Yaskawa INFORM job: X4-SCHODKI_ZEW.JBI

/JOB
//NAME X4-SCHODKI_ZEW
//POS
///NPOS 247,247,247,10,0,0
///TOOL 0
///POSTYPE PULSE
///PULSE
C00000=-21160,-126487,-99095,-6220,53097,-19917
C00001=-122314,-84956,-84267,-5758,65294,-20346
C00002=-113867,-2788,-32259,-11364,77586,20622
C00003=-111699,9606,-11794,-12514,71800,21939
C00004=-110873,16102,-4909,-12893,71047,22311
C00005=-111426,18220,-2948,-12689,70847,22135
C00006=-111334,17863,-3281,-12723,70881,22164
C00007=-111334,17842,-1921,-12786,70054,22254
C00008=-111688,13758,-7042,-12574,71029,22022
C00009=-137921,23655,2193,26065,80546,-13065
C00010=-138187,30095,8478,26164,80127,-13260
C00011=-137141,31636,10013,25924,79665,-12972
C00012=-137283,31426,9804,25956,79727,-13011
C00013=-137283,31447,11085,26011,79025,-13166
C00014=-137811,24810,3269,26040,80453,-13045
C00015=-130093,15204,-5597,17076,73087,-3422
C00016=-130254,16762,-4164,17139,73044,-3486
C00017=-130499,11823,-8660,17205,73314,-3535
C00018=-136657,16032,-4835,19303,74485,-5576
C00019=-136779,34044,12201,19450,73350,-5806
C00020=-136367,37287,16065,19383,72578,-5782
C00021=-135529,38270,17077,19116,72272,-5524
C00022=-135735,38345,17156,19186,72312,-5593
C00023=-135735,38391,18179,19247,71738,-5687
C00024=-136093,38073,17157,19317,72259,-5733
C00025=-136821,38987,18103,19565,72324,-5991
C00026=-137234,41236,20445,19732,72152,-6174
C00027=-137468,37941,16529,19737,72884,-6137
C00028=-139273,33119,8814,10616,74138,-14432
C00029=-138400,39162,15428,10360,73077,-14220
C00030=-137624,40756,17090,10099,72782,-13973
C00031=-137810,40443,16764,10163,72844,-14033
C00032=-137810,40460,18419,10216,71849,-14119
C00033=-138377,33107,10032,10341,73283,-14197
C00034=-129933,32626,9546,-1459,71562,-3103
C00035=-130107,34413,11352,-1398,71367,-3162
C00036=-130344,28976,5916,-1305,71915,-3250
C00037=-134876,30968,7890,396,71698,-4822
C00038=-142592,70732,50995,12851,68399,-16892
C00039=-141830,71409,51797,12602,68137,-16639
C00040=-142006,70894,51186,12652,68274,-16689
C00041=-142006,71149,52557,12712,67578,-16765
C00042=-142006,71007,51815,12679,67954,-16725
C00043=-142747,76515,58410,13043,66871,-17119
C00044=-142702,66110,44987,12780,69711,-16790
C00045=-130401,22900,-3912,-9781,74013,-14096
C00046=-130750,-77898,-76934,-10038,67211,-13654
C00047=-128341,-94500,-64478,-15665,37561,-8814
C00048=-125354,-34494,-33676,-16070,41961,-8103
C00049=-123908,-22688,-35224,7311,60763,-8117
C00050=-115329,1774,-22996,8583,68206,-33205
C00051=-113811,6923,-16554,7934,66753,-32769
C00052=-112938,8598,-15088,7517,66630,-32466
C00053=-113357,7607,-15958,7718,66694,-32611
C00054=-113357,7474,-14642,7767,65823,-32669
C00055=-113357,7562,-15559,7732,66427,-32629
C00056=-114674,8046,-17033,9196,71995,-10105
C00057=-114277,9137,-16073,9034,71921,-9973
C00058=-114994,10710,-14679,9331,71949,-10219
C00059=-115929,5782,-19714,10610,72890,-11247
C00060=-114914,9168,-18033,20160,83408,-25507
C00061=-114509,10465,-16323,20060,82947,-25443
C00062=-114509,10278,-15209,20089,82211,-25564
C00063=-114509,10430,-16126,20066,82816,-25464
C00064=-113574,12027,-14696,19812,82540,-25184
C00065=-113966,9476,-16971,19916,82715,-25292
C00066=-109195,41890,2270,19889,88323,-22522
C00067=-109420,41611,2136,14547,83651,-24420
C00068=-109633,43097,3705,14621,83493,-24508
C00069=-110073,47498,8361,9922,80898,-20177
C00070=-110340,48514,8983,10012,81065,-20250
C00071=-109875,50139,10594,6927,80049,-17487
C00072=-111642,41129,-2073,7513,83338,-17864
C00073=-120740,-4591,-30289,15267,55452,-23675
C00074=-120758,-111403,-89341,20679,37744,-27189
C00075=-120758,-111403,-89341,20679,37744,-27189
C00076=-97140,-41370,-74515,-11864,90116,15742
C00077=-93918,-16818,-51601,-15265,90472,19448
C00078=-96838,-21310,-54909,-14446,89719,18600
C00079=-97144,-22320,-55662,-14359,89616,18514
C00080=-98771,-24881,-57497,-13895,89173,18041
C00081=-115828,-29996,-61044,7286,86100,-2495
C00082=-121364,-24267,-57094,13933,89260,-9154
C00083=-125064,-13370,-49143,14990,90552,-10191
C00084=-125209,-12228,-48362,15033,90681,-10222
C00085=-127775,-3453,-41245,15747,91251,-10973
C00086=-117906,-11103,-47413,1372,86513,3179
C00087=-107817,-4833,-42392,-13913,90158,17947
C00088=-111065,-8601,-45456,-12965,89620,16971
C00089=-111228,-9142,-45834,-12917,89553,16926
C00090=-113235,-11504,-47787,-12324,89257,16321
C00091=-116129,-16038,-53218,-11461,89860,15351
C00092=-132129,3503,-37461,-731,88042,5165
C00093=-134330,9298,-30541,1308,86617,3236
C00094=-133591,9704,-30242,1064,86631,3463
C00095=-133365,10194,-29830,989,86627,3533
C00096=-132997,13157,-27039,5636,86965,-851
C00097=-131112,-12606,-50888,7793,88905,-29033
C00098=-129834,-10886,-48018,7386,87922,-28697
C00099=-133242,1411,-38107,8469,88444,-29724
C00100=-133268,2556,-37251,8479,88508,-29727
C00101=-132895,14601,-26523,2898,86979,-24450
C00102=-133144,15447,-25750,2979,86944,-24527
C00103=-133588,9909,-35564,3125,90148,-24585
C00104=-114600,-38617,-66572,-24501,76796,-21744
C00105=-88804,-102668,-113384,-34072,81784,-13502
C00106=3643,-76224,-106676,19950,71810,76872
C00107=6047,-95755,-92046,-14751,98253,9605
C00108=8024,-164446,-133802,-16041,6272,12396
C00109=8024,-164446,-133802,-16041,6272,12396
C00110=80911,-131071,-112390,-19160,57527,-4768
C00111=107387,-112645,-89313,-18613,48039,-3448
C00112=120529,-94925,-67119,-18087,38914,-2179
C00113=119158,-22093,-21003,-8683,62714,-5793
C00114=120616,-13235,-11129,-9376,61371,-5124
C00115=120244,-10241,-8815,-9223,61441,-5272
C00116=120242,-11093,-9478,-9225,61411,-5270
C00117=120242,-10458,-7028,-9331,60244,-5174
C00118=120224,-17007,-14555,-9215,61493,-5286
C00119=122889,-18524,910,-53470,54044,-6110
C00120=122847,-15690,3005,-53366,54123,-6195
C00121=122811,-12986,5045,-53281,54183,-6262
C00122=122821,-13724,4484,-53302,54168,-6245
C00123=122821,-12957,6355,-53740,53705,-5906
C00124=125895,-21581,-2992,-53539,56263,-5738
C00125=123923,-36868,-26996,-37261,61302,-5894
C00126=108816,-52753,-53811,-10212,62008,-9374
C00127=96034,-45136,-47055,9675,61622,-25160
C00128=97205,-43220,-45890,9111,61748,-24699
C00129=96974,-43470,-46044,9221,61740,-24787
C00130=96974,-43222,-44278,9303,60791,-24865
C00131=96448,-45521,-47615,9470,61714,-24990
C00132=118629,-40101,-48504,-12157,74776,12413
C00133=119364,-34097,-44083,-12359,75244,12623
C00134=118100,-32224,-42841,-11965,75251,12181
C00135=118253,-32582,-43080,-12015,75236,12237
C00136=118253,-32540,-41664,-12057,74406,12319
C00137=118721,-32602,-42752,-12165,75101,12411
C00138=116137,-37716,-46090,-11401,74165,11593
C00139=108993,-39238,-47060,-3979,71836,3847
C00140=109761,-37600,-46019,-4238,72074,4108
C00141=108993,-39238,-47060,-3979,71836,3847
C00142=117414,-43467,-49690,-6866,71847,6805
C00143=120406,-23125,-36428,-7781,74390,7697
C00144=120412,-21128,-34805,-7781,74419,7698
C00145=119620,-19753,-33804,-7516,74437,7425
C00146=119849,-20298,-34202,-7592,74423,7506
C00147=119849,-20300,-33096,-7616,73750,7551
C00148=119849,-20302,-33703,-7602,74119,7528
C00149=120845,-19874,-33391,-7929,74241,7866
C00150=121446,-18122,-32105,-8123,74405,8066
C00151=121464,-22241,-35587,-8130,74432,8070
C00152=122270,-32243,-42159,4732,69932,24573
C00153=121378,-24903,-37120,5049,70656,24286
C00154=120376,-23507,-36128,5424,70830,23939
C00155=120533,-24190,-36613,5366,70768,23993
C00156=120533,-24175,-35602,5386,70155,23966
C00157=120148,-30314,-42064,5504,71001,23867
C00158=110805,-25383,-38662,15109,74916,14576
C00159=111818,-22665,-36734,14771,74934,14940
C00160=111748,-27369,-40047,14817,74581,14871
C00161=119775,-28434,-40781,12151,73173,17551
C00162=124224,-1084,-19915,10540,73751,19166
C00163=130157,198,-18683,-209,73628,24476
C00164=130157,158,-17341,-210,72780,24477
C00165=130157,185,-18394,-210,73442,24477
C00166=129196,1421,-17357,132,73439,24146
C00167=130157,185,-18394,-210,73442,24477
C00168=122787,3680,-15441,12656,76349,11624
C00169=123743,5439,-13926,12357,76179,11938
C00170=123109,1410,-18093,12531,76759,11776
C00171=126751,-18741,-32489,13679,66636,29547
C00172=131594,-6512,-22252,11541,65879,31250
C00173=135627,-1986,-17513,3780,65616,32121
C00174=135627,-1956,-16347,3801,64914,32097
C00175=135627,-1986,-17486,3780,65599,32120
C00176=134800,-891,-16582,4152,65645,31822
C00177=135627,-1986,-17486,3780,65599,32120
C00178=122949,-12611,-24589,22132,67603,15841
C00179=121506,-8744,-21577,22663,68115,15387
C00180=122081,-6475,-19773,22437,68011,15585
C00181=121506,-8744,-21577,22663,68115,15387
C00182=127706,-12999,-26066,20142,67056,17565
C00183=136075,11793,-4386,8081,62286,35157
C00184=136075,11856,-3257,8130,61628,35109
C00185=136075,11798,-4304,8086,62236,35152
C00186=136366,13707,-2741,6760,62424,35173
C00187=136075,11798,-4304,8086,62236,35152
C00188=131305,-10305,-23416,10361,63176,33430
C00189=168291,-111367,-82610,-9688,47305,48503
C00190=206286,-74639,-65979,-25452,64014,61826
C00191=159660,-110455,-93035,-14572,38895,45711
C00192=139772,-9678,-45421,-20416,66544,-77404
C00193=128522,-26109,-48700,-36268,57340,-84657
C00194=119767,-9340,-33749,-20588,54929,-87055
C00195=118381,-12869,-36453,-19680,54464,-87541
C00196=118069,-13852,-36761,-19540,54093,-87599
C00197=119978,-17814,-39706,-30625,59015,-81414
C00198=119898,-18805,-40392,-30604,58911,-81418
C00199=117451,-25837,-45359,-31771,59062,-80695
C00200=122977,-25509,-47564,-34287,62428,-79397
C00201=137466,-21144,-46854,-40649,69913,-75869
C00202=196853,-39310,-56838,-56279,98183,-62272
C00203=239125,-37728,-55833,-56309,98295,-62347
C00204=198880,-64017,-70083,-47949,71692,22240
C00205=95782,-63494,-66422,9583,64100,-25040
C00206=96608,-32442,-40990,7123,69750,-24476
C00207=99153,-41436,-44893,7278,64322,-23821
C00208=98934,-42045,-45261,7777,64334,-23890
C00209=100370,-44106,-46526,7182,63922,-23380
C00210=119741,-40174,-44096,-19149,69535,-259
C00211=121592,-27553,-38534,-18093,79240,10876
C00212=125227,-17250,-31142,-18927,80757,11935
C00213=125393,-15914,-30142,-18963,80861,11977
C00214=127846,-8061,-24015,-19516,81680,12716
C00215=119795,-17677,-31449,-8017,74335,-710
C00216=108325,-15786,-29976,9492,74890,-18554
C00217=111630,-19800,-33189,8434,74445,-17438
C00218=111755,-20573,-33754,8397,74383,-17399
C00219=113687,-22438,-34957,7772,73974,-16756
C00220=117056,-24250,-37509,6639,74313,-15568
C00221=128480,-979,-19969,3779,76440,-7427
C00222=129844,2675,-15882,3356,75744,-6982
C00223=129268,3108,-15627,2949,75760,-6545
C00224=129028,3528,-15269,3025,75765,-6627
C00225=129576,5579,-13546,-2876,75741,-370
C00226=130057,-3886,-22978,-3018,76699,-230
C00227=122913,-28792,-41505,-1480,73376,7564
C00228=125274,-18849,-33719,-4896,77191,17730
C00229=131975,-10313,-25549,-10610,74903,19808
C00230=132069,-9167,-24748,-10635,75011,19832
C00231=135966,6668,-11544,-11862,75556,21141
C00232=130236,2592,-15119,-2350,73160,11427
C00233=128403,-11609,-30449,-1692,75251,10764
C00234=112588,-48510,-57222,11111,73491,6010
C00235=118900,-27089,-23855,-4947,60648,-6067
C00236=130292,-938,239,-22775,68727,4409
C00237=117379,-19874,-3208,-40401,48526,-8648
C00238=111452,-18537,-670,-42583,47269,-4687
C00239=115600,-23691,-9256,-36668,53200,-7502
C00240=123114,-34014,-31898,-14023,63529,-7414
C00241=103776,-61917,-65189,16989,73535,3120
C00242=77625,-115928,-93453,24842,70557,-7280
C00243=80911,-131071,-112390,-19160,57527,-4768
C00244=8024,-164446,-133802,-16041,6272,12396
C00245=8024,-164446,-133802,-16041,6272,12396
C00246=3643,-76224,-106676,19950,71810,76872
BC00000=277659,673923,172124
BC00001=328197,693320,172124
BC00002=328196,693321,172121
BC00003=328196,693321,172121
BC00004=328196,693321,172121
BC00005=328196,693321,172121
BC00006=328196,693321,172121
BC00007=328196,693321,172121
BC00008=328196,693321,172121
BC00009=328196,693321,172121
BC00010=328196,693321,172121
BC00011=328196,693321,172121
BC00012=328196,693321,172121
BC00013=328196,693321,172121
BC00014=328196,693321,172121
BC00015=328196,693321,172121
BC00016=328196,693321,172121
BC00017=328196,693321,172121
BC00018=328196,693321,172121
BC00019=328196,693321,172121
BC00020=328196,693321,172121
BC00021=328196,693321,172121
BC00022=328196,693321,172121
BC00023=328196,693321,172121
BC00024=328196,693321,172121
BC00025=328196,693321,172121
BC00026=328196,693321,172121
BC00027=328196,693321,172121
BC00028=328196,693321,172121
BC00029=328196,693321,172121
BC00030=328196,693321,172121
BC00031=328196,693321,172121
BC00032=328196,693321,172121
BC00033=328196,693321,172121
BC00034=328196,693321,172121
BC00035=328196,693321,172121
BC00036=328196,693321,172121
BC00037=328196,693321,172121
BC00038=328196,693321,172121
BC00039=328196,693321,172121
BC00040=328196,693321,172121
BC00041=328196,693321,172121
BC00042=328196,693321,172121
BC00043=328196,693321,172121
BC00044=328196,693321,172121
BC00045=328196,693321,172121
BC00046=328196,693321,172121
BC00047=194432,688081,172121
BC00048=194432,688081,172121
BC00049=173327,765103,172121
BC00050=173327,765103,140855
BC00051=173327,765103,140855
BC00052=173327,765103,140855
BC00053=173327,765103,140855
BC00054=173327,765103,140855
BC00055=173327,765103,140855
BC00056=173327,765103,140855
BC00057=173327,765103,140855
BC00058=173327,765103,140855
BC00059=173327,765103,140855
BC00060=173327,765103,140855
BC00061=173327,765103,140855
BC00062=173327,765103,140855
BC00063=173327,765103,140855
BC00064=173327,765103,140855
BC00065=173327,765103,140855
BC00066=158508,737843,59363
BC00067=158508,737843,59363
BC00068=158508,737843,59363
BC00069=158508,737843,59363
BC00070=158508,737843,59363
BC00071=158508,737843,59363
BC00072=158508,737843,59363
BC00073=158508,737843,59363
BC00074=158508,682152,59363
BC00075=293322,682152,59363
BC00076=293321,752433,59360
BC00077=293321,752433,59360
BC00078=293321,752433,59360
BC00079=293321,752433,59360
BC00080=293321,752433,59360
BC00081=293321,752433,59360
BC00082=293321,752433,59360
BC00083=293321,752433,59360
BC00084=293321,752433,59360
BC00085=293321,752433,59360
BC00086=293321,752433,59360
BC00087=293321,752433,59360
BC00088=293321,752433,59360
BC00089=293321,752433,59360
BC00090=293321,752433,59360
BC00091=293321,752433,59360
BC00092=293321,752433,59360
BC00093=293321,752433,59360
BC00094=293321,752433,59360
BC00095=293321,752433,59360
BC00096=293321,752433,59360
BC00097=293321,752433,59360
BC00098=293321,752433,59360
BC00099=293321,752433,59360
BC00100=293321,752433,59360
BC00101=293321,752433,59360
BC00102=293321,752433,59360
BC00103=293321,752433,59360
BC00104=293321,752433,59360
BC00105=293321,698561,59360
BC00106=199464,674570,1075173
BC00107=95044,675039,919146
BC00108=95044,675039,1075229
BC00109=235813,1345575,1075229
BC00110=291733,1363613,501241
BC00111=295042,1365829,344881
BC00112=288108,1367960,194507
BC00113=288108,1367960,194507
BC00114=288108,1367960,194507
BC00115=288108,1367960,194507
BC00116=288108,1367960,194507
BC00117=288108,1367960,194507
BC00118=288108,1367960,194507
BC00119=288108,1367960,194507
BC00120=288108,1367960,194507
BC00121=288108,1367960,194507
BC00122=288108,1367960,194507
BC00123=288108,1367960,194507
BC00124=288108,1367960,194507
BC00125=288108,1367445,194507
BC00126=288108,1366688,194507
BC00127=288109,1366690,194504
BC00128=288109,1366690,194504
BC00129=288109,1366690,194504
BC00130=288109,1366690,194504
BC00131=288109,1366690,194504
BC00132=288109,1366690,194504
BC00133=288109,1366690,194504
BC00134=288109,1366690,194504
BC00135=288109,1366690,194504
BC00136=288109,1366690,194504
BC00137=288109,1366690,194504
BC00138=288109,1366690,194504
BC00139=288109,1366690,194504
BC00140=288109,1366690,194504
BC00141=288109,1366690,194504
BC00142=288109,1366690,194504
BC00143=288109,1366690,194504
BC00144=288109,1366690,194504
BC00145=288109,1366690,194504
BC00146=288109,1366690,194504
BC00147=288109,1366690,194504
BC00148=288109,1366690,194504
BC00149=288109,1366690,194504
BC00150=288109,1366690,194504
BC00151=288109,1366690,194504
BC00152=288109,1366690,194504
BC00153=288109,1366690,194504
BC00154=288109,1366690,194504
BC00155=288109,1366690,194504
BC00156=288109,1366690,194504
BC00157=288109,1366690,194504
BC00158=288109,1366690,194504
BC00159=288109,1366690,194504
BC00160=288109,1366690,194504
BC00161=288109,1366690,194504
BC00162=288109,1366690,194504
BC00163=288109,1366690,194504
BC00164=288109,1366690,194504
BC00165=288109,1366690,194504
BC00166=288109,1366690,194504
BC00167=288109,1366690,194504
BC00168=288109,1366690,194504
BC00169=288109,1366690,194504
BC00170=288109,1366690,194504
BC00171=288109,1366690,194504
BC00172=288109,1366690,194504
BC00173=288109,1366690,194504
BC00174=288109,1366690,194504
BC00175=288109,1366690,194504
BC00176=288109,1366690,194504
BC00177=288109,1366690,194504
BC00178=288109,1366690,194504
BC00179=288109,1366690,194504
BC00180=288109,1366690,194504
BC00181=288109,1366690,194504
BC00182=288109,1366690,194504
BC00183=288109,1366690,194504
BC00184=288109,1366690,194504
BC00185=288109,1366690,194504
BC00186=288109,1366690,194504
BC00187=288109,1366690,194504
BC00188=288109,1366690,194504
BC00189=362373,1366690,194504
BC00190=212912,1366690,52238
BC00191=212912,1366690,52238
BC00192=212912,1366690,52238
BC00193=181372,1351458,52238
BC00194=181372,1351458,52238
BC00195=181372,1351458,52238
BC00196=181372,1351458,52238
BC00197=181372,1351458,52238
BC00198=181372,1351458,52238
BC00199=181372,1351458,52238
BC00200=181372,1351458,52238
BC00201=181372,1351458,52238
BC00202=258948,1351458,52238
BC00203=397724,1351458,84656
BC00204=397724,1351458,84656
BC00205=288109,1366690,194504
BC00206=288109,1366690,194504
BC00207=288109,1366690,194504
BC00208=288109,1366690,194504
BC00209=288109,1366690,194504
BC00210=288109,1366690,194504
BC00211=288109,1366690,194504
BC00212=288109,1366690,194504
BC00213=288109,1366690,194504
BC00214=288109,1366690,194504
BC00215=288109,1366690,194504
BC00216=288109,1366690,194504
BC00217=288109,1366690,194504
BC00218=288109,1366690,194504
BC00219=288109,1366690,194504
BC00220=288109,1366690,194504
BC00221=288109,1366690,194504
BC00222=288109,1366690,194504
BC00223=288109,1366690,194504
BC00224=288109,1366690,194504
BC00225=288109,1366690,194504
BC00226=288109,1366690,194504
BC00227=288109,1366690,194504
BC00228=288109,1366690,194504
BC00229=288109,1366690,194504
BC00230=288109,1366690,194504
BC00231=288109,1366690,194504
BC00232=288109,1366690,194504
BC00233=288109,1366690,194504
BC00234=288109,1366690,194504
BC00235=288109,1366690,194504
BC00236=288109,1366690,194504
BC00237=288109,1366690,194504
BC00238=288109,1366690,194504
BC00239=288109,1366690,194504
BC00240=288109,1366690,194504
BC00241=288109,1366690,194504
BC00242=288109,1366690,194504
BC00243=269895,1363613,501241
BC00244=235813,1345575,1075229
BC00245=95044,675039,1075229
BC00246=199464,674570,1075173
EC00000=-798156,0
EC00001=-798156,0
EC00002=-798153,-1
EC00003=-798153,-1
EC00004=-798153,-1
EC00005=-798153,-1
EC00006=-798153,-1
EC00007=-798153,-1
EC00008=-798153,-1
EC00009=-798153,-1
EC00010=-798153,-1
EC00011=-798153,-1
EC00012=-798153,-1
EC00013=-798153,-1
EC00014=-798153,-1
EC00015=-798153,-1
EC00016=-798153,-1
EC00017=-798153,-1
EC00018=-798153,-1
EC00019=-798153,-1
EC00020=-798153,-1
EC00021=-798153,-1
EC00022=-798153,-1
EC00023=-798153,-1
EC00024=-798153,-1
EC00025=-798153,-1
EC00026=-798153,-1
EC00027=-798153,-1
EC00028=-798153,-1
EC00029=-798153,-1
EC00030=-798153,-1
EC00031=-798153,-1
EC00032=-798153,-1
EC00033=-798153,-1
EC00034=-798153,-1
EC00035=-798153,-1
EC00036=-798153,-1
EC00037=-798153,-1
EC00038=-798153,-1
EC00039=-798153,-1
EC00040=-798153,-1
EC00041=-798153,-1
EC00042=-798153,-1
EC00043=-798153,-1
EC00044=-798153,-1
EC00045=-798153,-1
EC00046=-798153,-1
EC00047=-798153,-1
EC00048=-798153,-1
EC00049=-798153,-1
EC00050=-798153,-1
EC00051=-798153,-1
EC00052=-798153,-1
EC00053=-798153,-1
EC00054=-798153,-1
EC00055=-798153,-1
EC00056=-798153,-1
EC00057=-798153,-1
EC00058=-798153,-1
EC00059=-798153,-1
EC00060=-798153,-1
EC00061=-798153,-1
EC00062=-798153,-1
EC00063=-798153,-1
EC00064=-798153,-1
EC00065=-798153,-1
EC00066=-798153,-1
EC00067=-798153,-1
EC00068=-798153,-1
EC00069=-798153,-1
EC00070=-798153,-1
EC00071=-798153,-1
EC00072=-798153,-1
EC00073=-798153,-1
EC00074=-798153,-1
EC00075=-798153,-1
EC00076=-798151,-2
EC00077=-798151,-2
EC00078=-798151,-2
EC00079=-798151,-2
EC00080=-798151,-2
EC00081=-798151,-2
EC00082=-798151,-2
EC00083=-798151,-2
EC00084=-798151,-2
EC00085=-798151,-2
EC00086=-798151,-2
EC00087=-798151,-2
EC00088=-798151,-2
EC00089=-798151,-2
EC00090=-798151,-2
EC00091=-798151,-2
EC00092=-798151,-2
EC00093=-798151,-2
EC00094=-798151,-2
EC00095=-798151,-2
EC00096=-798151,-2
EC00097=-798151,-2
EC00098=-798151,-2
EC00099=-798151,-2
EC00100=-798151,-2
EC00101=-798151,-2
EC00102=-798151,-2
EC00103=-798151,-2
EC00104=-798151,-2
EC00105=-798151,-2
EC00106=-798151,-2
EC00107=-798156,0
EC00108=798156,0
EC00109=798156,0
EC00110=798156,0
EC00111=798156,0
EC00112=798156,0
EC00113=798156,0
EC00114=798156,0
EC00115=798156,0
EC00116=798156,0
EC00117=798156,0
EC00118=798156,0
EC00119=798156,0
EC00120=798156,0
EC00121=798156,0
EC00122=798156,0
EC00123=798156,0
EC00124=798156,0
EC00125=798156,0
EC00126=798156,0
EC00127=798155,0
EC00128=798155,0
EC00129=798155,0
EC00130=798155,0
EC00131=798155,0
EC00132=798155,0
EC00133=798155,0
EC00134=798155,0
EC00135=798155,0
EC00136=798155,0
EC00137=798155,0
EC00138=798155,0
EC00139=798155,0
EC00140=798155,0
EC00141=798155,0
EC00142=798155,0
EC00143=798155,0
EC00144=798155,0
EC00145=798155,0
EC00146=798155,0
EC00147=798155,0
EC00148=798155,0
EC00149=798155,0
EC00150=798155,0
EC00151=798155,0
EC00152=798155,0
EC00153=798155,0
EC00154=798155,0
EC00155=798155,0
EC00156=798155,0
EC00157=798155,0
EC00158=798155,0
EC00159=798155,0
EC00160=798155,0
EC00161=798155,0
EC00162=798155,0
EC00163=798155,0
EC00164=798155,0
EC00165=798155,0
EC00166=798155,0
EC00167=798155,0
EC00168=798155,0
EC00169=798155,0
EC00170=798155,0
EC00171=798155,0
EC00172=798155,0
EC00173=798155,0
EC00174=798155,0
EC00175=798155,0
EC00176=798155,0
EC00177=798155,0
EC00178=798155,0
EC00179=798155,0
EC00180=798155,0
EC00181=798155,0
EC00182=798155,0
EC00183=798155,0
EC00184=798155,0
EC00185=798155,0
EC00186=798155,0
EC00187=798155,0
EC00188=798155,0
EC00189=798155,0
EC00190=798155,0
EC00191=798155,0
EC00192=798155,0
EC00193=798155,0
EC00194=798155,0
EC00195=798155,0
EC00196=798155,0
EC00197=798155,0
EC00198=798155,0
EC00199=798155,0
EC00200=798155,0
EC00201=798155,0
EC00202=798155,0
EC00203=798155,0
EC00204=798155,0
EC00205=798155,0
EC00206=798155,0
EC00207=798155,0
EC00208=798155,0
EC00209=798155,0
EC00210=798155,0
EC00211=798155,0
EC00212=798155,0
EC00213=798155,0
EC00214=798155,0
EC00215=798155,0
EC00216=798155,0
EC00217=798155,0
EC00218=798155,0
EC00219=798155,0
EC00220=798155,0
EC00221=798155,0
EC00222=798155,0
EC00223=798155,0
EC00224=798155,0
EC00225=798155,0
EC00226=798155,0
EC00227=798155,0
EC00228=798155,0
EC00229=798155,0
EC00230=798155,0
EC00231=798155,0
EC00232=798155,0
EC00233=798155,0
EC00234=798155,0
EC00235=798155,0
EC00236=798155,0
EC00237=798155,0
EC00238=798155,0
EC00239=798155,0
EC00240=798155,0
EC00241=798155,0
EC00242=798155,0
EC00243=798156,0
EC00244=798156,0
EC00245=798156,0
EC00246=798156,0
///POSTYPE BASE
///RECTAN
///RCONF 0,0,0,0,0,0,0,0,0,0,0,0,0,0,0,0,0,0,0,0,0,0,0,0
P00006=0.000,0.000,0.000,0.0000,0.0000,0.0000
P00021=1.195,-1.322,-3.236,0.0000,0.0000,0.0000
P00022=0.222,-3.123,-1.508,0.0000,0.0000,0.0000
P00023=0.143,-0.036,0.682,0.0000,0.0000,0.0000
P00024=0.145,-0.552,1.326,0.0000,0.0000,0.0000
P00025=-2.003,0.006,0.728,0.0000,0.0000,0.0000
P00026=0.562,-0.002,-0.337,0.0000,0.0000,0.0000
P00027=-0.746,0.015,-9.096,0.0000,0.0000,0.0000
P00030=5.926,-4.294,-1.390,0.0000,0.0000,0.0000
P00031=1.853,-0.001,-1.549,0.0000,0.0000,0.0000
//INST
///DATE 2024/04/14 21:21
///ATTR SC,RW
///GROUP1 RB1,BS1
///GROUP2 ST1
NOP
MOVJ C00000 BC00000 VJ=100.00  +MOVJ EC00000 VJ=100.00
MOVJ C00001 BC00001 VJ=100.00  +MOVJ EC00001 VJ=100.00
MOVJ C00002 BC00002 VJ=100.00  +MOVJ EC00002 VJ=100.00
SMOVL C00003 BC00003 V=833.3  +MOVJ EC00003
SMOVL C00004 BC00004 V=166.7  +MOVJ EC00004
SREFP 3 C00005 BC00005  +REFP EC00005
CALL JOB:SEARCH-R1-S13D
SET P021 P006
SFTON3D P021
SMOVL C00006 BC00006 V=166.7  +MOVJ EC00006
SREFP 3 C00007 BC00007  +REFP EC00007
CALL JOB:SEARCH-R1-S13D
SET P021 P006
SFTON3D P021
SMOVL C00008 BC00008 V=166.7  +MOVJ EC00008
SFTOF3D
SMOVL C00009 BC00009 V=833.3  +MOVJ EC00009
SMOVL C00010 BC00010 V=166.7  +MOVJ EC00010
SREFP 3 C00011 BC00011  +REFP EC00011
CALL JOB:SEARCH-R1-S13D
SET P022 P006
SFTON3D P022
SMOVL C00012 BC00012 V=166.7  +MOVJ EC00012
SREFP 3 C00013 BC00013  +REFP EC00013
CALL JOB:SEARCH-R1-S13D
SET P022 P006
SFTON3D P022
SMOVL C00014 BC00014 V=166.7  +MOVJ EC00014
SMOVL C00015 BC00015 V=166.7  +MOVJ EC00015
SREFP 3 C00016 BC00016  +REFP EC00016
CALL JOB:SEARCH-R1-S13D
SET P022 P006
SFTON3D P022
SMOVL C00017 BC00017 V=166.7  +MOVJ EC00017
SFTOF3D
SMOVL C00018 BC00018 V=500.0  +MOVJ EC00018
SMOVL C00019 BC00019 V=500.0  +MOVJ EC00019
SMOVL C00020 BC00020 V=166.7  +MOVJ EC00020
SREFP 3 C00021 BC00021  +REFP EC00021
CALL JOB:SEARCH-R1-S13D
SET P023 P006
SFTON3D P023
SMOVL C00022 BC00022 V=166.7  +MOVJ EC00022
SREFP 3 C00023 BC00023  +REFP EC00023
CALL JOB:SEARCH-R1-S13D
SET P023 P006
SFTON3D P023
SMOVL C00024 BC00024 V=166.7  +MOVJ EC00024
SMOVL C00025 BC00025 V=166.7  +MOVJ EC00025
SREFP 3 C00026 BC00026  +REFP EC00026
CALL JOB:SEARCH-R1-S13D
SET P023 P006
SFTON3D P023
SMOVL C00027 BC00027 V=166.7  +MOVJ EC00027
SFTOF3D
SMOVL C00028 BC00028 V=333.3  +MOVJ EC00028
SMOVL C00029 BC00029 V=166.7  +MOVJ EC00029
SREFP 3 C00030 BC00030  +REFP EC00030
CALL JOB:SEARCH-R1-S13D
SET P024 P006
SFTON3D P024
SMOVL C00031 BC00031 V=166.7  +MOVJ EC00031
SREFP 3 C00032 BC00032  +REFP EC00032
CALL JOB:SEARCH-R1-S13D
SET P024 P006
SFTON3D P024
SMOVL C00033 BC00033 V=166.7  +MOVJ EC00033
SMOVL C00034 BC00034 V=166.7  +MOVJ EC00034
SREFP 3 C00035 BC00035  +REFP EC00035
CALL JOB:SEARCH-R1-S13D
SET P024 P006
SFTON3D P024
SMOVL C00036 BC00036 V=166.7  +MOVJ EC00036
SFTOF3D
SMOVL C00037 BC00037 V=333.3  +MOVJ EC00037
SMOVL C00038 BC00038 V=166.7  +MOVJ EC00038
SREFP 3 C00039 BC00039  +REFP EC00039
CALL JOB:SEARCH-R1-S13D
SET P025 P006
SFTON3D P025
SMOVL C00040 BC00040 V=166.7  +MOVJ EC00040
SREFP 3 C00041 BC00041  +REFP EC00041
CALL JOB:SEARCH-R1-S13D
SET P025 P006
SFTON3D P025
SMOVL C00042 BC00042 V=166.7  +MOVJ EC00042
SREFP 3 C00043 BC00043  +REFP EC00043
CALL JOB:SEARCH-R1-S13D
SET P025 P006
SFTON3D P025
SMOVL C00044 BC00044 V=166.7  +MOVJ EC00044
SFTOF3D
SMOVL C00045 BC00045 V=333.3  +MOVJ EC00045
SMOVL C00046 BC00046 V=1000.0  +MOVJ EC00046
SMOVL C00047 BC00047 V=1000.0  +MOVJ EC00047
SMOVL C00048 BC00048 V=1000.0  +MOVJ EC00048
SMOVL C00049 BC00049 V=666.7  +MOVJ EC00049
SMOVL C00050 BC00050 V=666.7  +MOVJ EC00050
SMOVL C00051 BC00051 V=166.7  +MOVJ EC00051
SREFP 3 C00052 BC00052  +REFP EC00052
CALL JOB:SEARCH-R1-S13D
SET P027 P006
SFTON3D P027
SMOVL C00053 BC00053 V=166.7  +MOVJ EC00053
SREFP 3 C00054 BC00054  +REFP EC00054
CALL JOB:SEARCH-R1-S13D
SET P027 P006
SFTON3D P027
SMOVL C00055 BC00055 V=166.7  +MOVJ EC00055
SMOVL C00056 BC00056 V=250.0  +MOVJ EC00056
SMOVL C00057 BC00057 V=250.0  +MOVJ EC00057
SREFP 3 C00058 BC00058  +REFP EC00058
CALL JOB:SEARCH-R1-S13D
SET P027 P006
SFTON3D P027
SMOVL C00059 BC00059 V=166.7  +MOVJ EC00059
SFTOF3D
SMOVL C00060 BC00060 V=250.0  +MOVJ EC00060
SMOVL C00061 BC00061 V=166.7  +MOVJ EC00061
SREFP 3 C00062 BC00062  +REFP EC00062
CALL JOB:SEARCH-R1-S13D
SET P026 P006
SFTON3D P026
SMOVL C00063 BC00063 V=166.7  +MOVJ EC00063
SREFP 3 C00064 BC00064  +REFP EC00064
CALL JOB:SEARCH-R1-S13D
SET P026 P006
SFTON3D P026
SMOVL C00065 BC00065 V=166.7  +MOVJ EC00065
MACRO1 MJ#(0) ARGF9
SMOVL C00066 BC00066 V=250.0  +MOVJ EC00066
ARCON
SMOVL C00067 BC00067 V=10.0  +MOVJ EC00067
SMOVL C00068 BC00068 V=10.0  +MOVJ EC00068
SFTON3D P027
SMOVL C00069 BC00069 V=10.0  +MOVJ EC00069
ARCOF
SMOVL C00070 BC00070 V=10.0  +MOVJ EC00070
ARCON
SMOVL C00071 BC00071 V=10.0  +MOVJ EC00071
ARCOF
SFTOF3D
SMOVL C00072 BC00072 V=250.0  +MOVJ EC00072
SMOVL C00073 BC00073 V=666.7  +MOVJ EC00073
SMOVL C00074 BC00074 V=666.7  +MOVJ EC00074
SMOVL C00075 BC00075 V=1000.0  +MOVJ EC00075
SMOVL C00076 BC00076 V=1000.0  +MOVJ EC00076
SFTON3D P021
SMOVL C00077 BC00077 V=166.7  +MOVJ EC00077
ARCON
SMOVL C00078 BC00078 V=10.0  +MOVJ EC00078
SFTON3D P022
SMOVL C00079 BC00079 V=10.0  +MOVJ EC00079
SMOVL C00080 BC00080 V=10.0  +MOVJ EC00080
SMOVL C00081 BC00081 V=10.0  +MOVJ EC00081
SMOVL C00082 BC00082 V=10.0  +MOVJ EC00082
SMOVL C00083 BC00083 V=10.0  +MOVJ EC00083
SMOVL C00084 BC00084 V=10.0  +MOVJ EC00084
SFTON3D P023
SMOVL C00085 BC00085 V=10.0  +MOVJ EC00085
SMOVL C00086 BC00086 V=10.0  +MOVJ EC00086
SMOVL C00087 BC00087 V=10.0  +MOVJ EC00087
SMOVL C00088 BC00088 V=10.0  +MOVJ EC00088
SFTON3D P024
SMOVL C00089 BC00089 V=10.0  +MOVJ EC00089
SMOVL C00090 BC00090 V=10.0  +MOVJ EC00090
ARCOF
SFTOF3D
SMOVL C00091 BC00091 V=250.0  +MOVJ EC00091
SMOVL C00092 BC00092 V=500.0  +MOVJ EC00092
SFTON3D P026
SMOVL C00093 BC00093 V=250.0  +MOVJ EC00093
ARCON
SMOVL C00094 BC00094 V=10.0  +MOVJ EC00094
SMOVL C00095 BC00095 V=10.0  +MOVJ EC00095
SFTON3D P025
SMOVL C00096 BC00096 V=10.0  +MOVJ EC00096
ARCOF
SFTOF3D
SMOVL C00097 BC00097 V=400.0  +MOVJ EC00097
SFTON3D P024
SMOVL C00098 BC00098 V=166.7  +MOVJ EC00098
ARCON
SMOVL C00099 BC00099 V=10.0  +MOVJ EC00099
SMOVL C00100 BC00100 V=10.0  +MOVJ EC00100
SFTON3D P025
SMOVL C00101 BC00101 V=10.0  +MOVJ EC00101
SMOVL C00102 BC00102 V=10.0  +MOVJ EC00102
ARCOF
SFTOF3D
SMOVL C00103 BC00103 V=250.0  +MOVJ EC00103
SMOVL C00104 BC00104 V=833.3  +MOVJ EC00104
MOVJ C00105 BC00105 VJ=100.00  +MOVJ EC00105 VJ=100.00
MOVJ C00106 BC00106 VJ=100.00  +MOVJ EC00106 VJ=100.00
CALL JOB:CLEAN-R1_KM_NEW
MOVJ C00107 BC00107 VJ=100.00  +MOVJ EC00107 VJ=100.00
MOVJ C00108 BC00108 VJ=100.00  +MOVJ EC00108 VJ=100.00
MOVJ C00109 BC00109 VJ=100.00  +MOVJ EC00109 VJ=100.00
'obrot
MOVJ C00110 BC00110 VJ=100.00  +MOVJ EC00110 VJ=100.00
MOVJ C00111 BC00111 VJ=100.00  +MOVJ EC00111 VJ=100.00
MOVJ C00112 BC00112 VJ=100.00  +MOVJ EC00112 VJ=100.00
SFTOF3D
SMOVL C00113 BC00113 V=500.0  +MOVJ EC00113
SMOVL C00114 BC00114 V=166.7  +MOVJ EC00114
SREFP 3 C00115 BC00115  +REFP EC00115
CALL JOB:SEARCH-R1-S13D
SET P030 P006
SFTON3D P030
SMOVL C00116 BC00116 V=166.7  +MOVJ EC00116
SREFP 3 C00117 BC00117  +REFP EC00117
CALL JOB:SEARCH-R1-S13D
SET P030 P006
SFTON3D P030
SMOVL C00118 BC00118 V=166.7  +MOVJ EC00118
SFTOF3D
SMOVL C00119 BC00119 V=500.0  +MOVJ EC00119
SMOVL C00120 BC00120 V=166.7  +MOVJ EC00120
SREFP 3 C00121 BC00121  +REFP EC00121
CALL JOB:SEARCH-R1-S13D
SET P031 P006
SFTON3D P031
SMOVL C00122 BC00122 V=166.7  +MOVJ EC00122
SREFP 3 C00123 BC00123  +REFP EC00123
CALL JOB:SEARCH-R1-S13D
SET P031 P006
SFTON3D P031
SMOVL C00124 BC00124 V=166.7  +MOVJ EC00124
SMOVL C00125 BC00125 V=416.7  +MOVJ EC00125
'Path S4271
SFTOF3D
MOVJ C00126 BC00126 VJ=50.00  +MOVJ EC00126 VJ=50.00
SMOVL C00127 BC00127 V=166.7  +MOVJ EC00127
SREFP 3 C00128 BC00128  +REFP EC00128
CALL JOB:SEARCH-R1-S13D
SET P021 P006
SFTON3D P021
SMOVL C00129 BC00129 V=166.7  +MOVJ EC00129
SREFP 3 C00130 BC00130  +REFP EC00130
CALL JOB:SEARCH-R1-S13D
SET P021 P006
SFTON3D P021
SMOVL C00131 BC00131 V=166.7  +MOVJ EC00131
SFTOF3D
SMOVL C00132 BC00132 V=833.3  +MOVJ EC00132
SMOVL C00133 BC00133 V=166.7  +MOVJ EC00133
SREFP 3 C00134 BC00134  +REFP EC00134
CALL JOB:SEARCH-R1-S13D
SET P022 P006
SFTON3D P022
SMOVL C00135 BC00135 V=166.7  +MOVJ EC00135
SREFP 3 C00136 BC00136  +REFP EC00136
CALL JOB:SEARCH-R1-S13D
SET P022 P006
SFTON3D P022
SMOVL C00137 BC00137 V=166.7  +MOVJ EC00137
SMOVL C00138 BC00138 V=166.7  +MOVJ EC00138
SMOVL C00139 BC00139 V=166.7  +MOVJ EC00139
SREFP 3 C00140 BC00140  +REFP EC00140
CALL JOB:SEARCH-R1-S13D
SET P022 P006
SFTON3D P022
SMOVL C00141 BC00141 V=166.7  +MOVJ EC00141
SFTOF3D
SMOVL C00142 BC00142 V=500.0  +MOVJ EC00142
SMOVL C00143 BC00143 V=500.0  +MOVJ EC00143
SMOVL C00144 BC00144 V=166.7  +MOVJ EC00144
SREFP 3 C00145 BC00145  +REFP EC00145
CALL JOB:SEARCH-R1-S13D
SET P023 P006
SFTON3D P023
SMOVL C00146 BC00146 V=166.7  +MOVJ EC00146
SREFP 3 C00147 BC00147  +REFP EC00147
CALL JOB:SEARCH-R1-S13D
SET P023 P006
SFTON3D P023
SMOVL C00148 BC00148 V=166.7  +MOVJ EC00148
SMOVL C00149 BC00149 V=166.7  +MOVJ EC00149
SREFP 3 C00150 BC00150  +REFP EC00150
CALL JOB:SEARCH-R1-S13D
SET P023 P006
SFTON3D P023
SMOVL C00151 BC00151 V=166.7  +MOVJ EC00151
SFTOF3D
SMOVL C00152 BC00152 V=333.3  +MOVJ EC00152
SMOVL C00153 BC00153 V=166.7  +MOVJ EC00153
SREFP 3 C00154 BC00154  +REFP EC00154
CALL JOB:SEARCH-R1-S13D
SET P024 P006
SFTON3D P024
SMOVL C00155 BC00155 V=166.7  +MOVJ EC00155
SREFP 3 C00156 BC00156  +REFP EC00156
CALL JOB:SEARCH-R1-S13D
SET P024 P006
SFTON3D P024
SMOVL C00157 BC00157 V=166.7  +MOVJ EC00157
SMOVL C00158 BC00158 V=166.7  +MOVJ EC00158
SREFP 3 C00159 BC00159  +REFP EC00159
CALL JOB:SEARCH-R1-S13D
SET P024 P006
SFTON3D P024
SMOVL C00160 BC00160 V=166.7  +MOVJ EC00160
SFTOF3D
SMOVL C00161 BC00161 V=333.3  +MOVJ EC00161
SMOVL C00162 BC00162 V=333.3  +MOVJ EC00162
SMOVL C00163 BC00163 V=166.7  +MOVJ EC00163
SREFP 3 C00164 BC00164  +REFP EC00164
CALL JOB:SEARCH-R1-S13D
SET P025 P006
SFTON3D P025
SMOVL C00165 BC00165 V=166.7  +MOVJ EC00165
SREFP 3 C00166 BC00166  +REFP EC00166
CALL JOB:SEARCH-R1-S13D
SET P025 P006
SFTON3D P025
SMOVL C00167 BC00167 V=166.7  +MOVJ EC00167
SMOVL C00168 BC00168 V=166.7  +MOVJ EC00168
SREFP 3 C00169 BC00169  +REFP EC00169
CALL JOB:SEARCH-R1-S13D
SET P025 P006
SFTON3D P025
SMOVL C00170 BC00170 V=166.7  +MOVJ EC00170
SFTOF3D
SMOVL C00171 BC00171 V=333.3  +MOVJ EC00171
SMOVL C00172 BC00172 V=1000.0  +MOVJ EC00172
SMOVL C00173 BC00173 V=166.7  +MOVJ EC00173
SREFP 3 C00174 BC00174  +REFP EC00174
CALL JOB:SEARCH-R1-S13D
SET P027 P006
SFTON3D P027
SMOVL C00175 BC00175 V=166.7  +MOVJ EC00175
SREFP 3 C00176 BC00176  +REFP EC00176
CALL JOB:SEARCH-R1-S13D
SET P027 P006
SFTON3D P027
SMOVL C00177 BC00177 V=166.7  +MOVJ EC00177
SMOVL C00178 BC00178 V=250.0  +MOVJ EC00178
SMOVL C00179 BC00179 V=250.0  +MOVJ EC00179
SREFP 3 C00180 BC00180  +REFP EC00180
CALL JOB:SEARCH-R1-S13D
SET P027 P006
SFTON3D P027
SMOVL C00181 BC00181 V=166.7  +MOVJ EC00181
SFTOF3D
SMOVL C00182 BC00182 V=250.0  +MOVJ EC00182
SMOVL C00183 BC00183 V=166.7  +MOVJ EC00183
SREFP 3 C00184 BC00184  +REFP EC00184
CALL JOB:SEARCH-R1-S13D
SET P026 P006
SFTON3D P026
SMOVL C00185 BC00185 V=166.7  +MOVJ EC00185
SREFP 3 C00186 BC00186  +REFP EC00186
CALL JOB:SEARCH-R1-S13D
SET P026 P006
SFTON3D P026
SMOVL C00187 BC00187 V=166.7  +MOVJ EC00187
SMOVL C00188 BC00188 V=166.7  +MOVJ EC00188
SFTOF3D
SMOVL C00189 BC00189 V=500.0  +MOVJ EC00189
SMOVL C00190 BC00190 V=500.0  +MOVJ EC00190
MOVJ C00191 BC00191 VJ=20.00  +MOVJ EC00191 VJ=20.00
MOVJ C00192 BC00192 VJ=20.00  +MOVJ EC00192 VJ=100.00
MOVJ C00193 BC00193 VJ=20.00  +MOVJ EC00193 VJ=20.00
MACRO1 MJ#(0) ARGF9
SFTON3D P026
SMOVL C00194 BC00194 V=250.0  +MOVJ EC00194
ARCON
SMOVL C00195 BC00195 V=10.0  +MOVJ EC00195
SMOVL C00196 BC00196 V=10.0  +MOVJ EC00196
SFTON3D P027
SMOVL C00197 BC00197 V=10.0  +MOVJ EC00197
SMOVL C00198 BC00198 V=10.0  +MOVJ EC00198
SMOVL C00199 BC00199 V=10.0  +MOVJ EC00199
ARCOF
SFTOF3D
SMOVL C00200 BC00200 V=250.0  +MOVJ EC00200
SMOVL C00201 BC00201 V=500.0  +MOVJ EC00201
SMOVL C00202 BC00202 V=666.7  +MOVJ EC00202
SMOVL C00203 BC00203 V=500.0  +MOVJ EC00203
MOVJ C00204 BC00204 VJ=20.00  +MOVJ EC00204 VJ=20.00
MOVJ C00205 BC00205 VJ=20.00  +MOVJ EC00205 VJ=20.00
SFTON3D P021
SMOVL C00206 BC00206 V=166.7  +MOVJ EC00206
ARCON
SMOVL C00207 BC00207 V=10.0  +MOVJ EC00207
SFTON3D P022
SMOVL C00208 BC00208 V=10.0  +MOVJ EC00208
SMOVL C00209 BC00209 V=10.0  +MOVJ EC00209
SMOVL C00210 BC00210 V=10.0  +MOVJ EC00210
SMOVL C00211 BC00211 V=10.0  +MOVJ EC00211
SMOVL C00212 BC00212 V=10.0  +MOVJ EC00212
SMOVL C00213 BC00213 V=10.0  +MOVJ EC00213
SFTON3D P023
SMOVL C00214 BC00214 V=10.0  +MOVJ EC00214
SMOVL C00215 BC00215 V=10.0  +MOVJ EC00215
SMOVL C00216 BC00216 V=10.0  +MOVJ EC00216
SMOVL C00217 BC00217 V=10.0  +MOVJ EC00217
SFTON3D P024
SMOVL C00218 BC00218 V=10.0  +MOVJ EC00218
SMOVL C00219 BC00219 V=10.0  +MOVJ EC00219
ARCOF
SFTOF3D
SMOVL C00220 BC00220 V=250.0  +MOVJ EC00220
SMOVL C00221 BC00221 V=500.0  +MOVJ EC00221
SFTON3D P026
SMOVL C00222 BC00222 V=250.0  +MOVJ EC00222
ARCON
SMOVL C00223 BC00223 V=10.0  +MOVJ EC00223
SMOVL C00224 BC00224 V=10.0  +MOVJ EC00224
SFTON3D P025
SMOVL C00225 BC00225 V=10.0  +MOVJ EC00225
ARCOF
SFTOF3D
SMOVL C00226 BC00226 V=400.0  +MOVJ EC00226
SMOVL C00227 BC00227 V=500.0  +MOVJ EC00227
SFTON3D P024
SMOVL C00228 BC00228 V=166.7  +MOVJ EC00228
ARCON
SMOVL C00229 BC00229 V=10.0  +MOVJ EC00229
SMOVL C00230 BC00230 V=10.0  +MOVJ EC00230
SFTON3D P025
SMOVL C00231 BC00231 V=10.0  +MOVJ EC00231
SMOVL C00232 BC00232 V=10.0  +MOVJ EC00232
ARCOF
SFTOF3D
SMOVL C00233 BC00233 V=250.0  +MOVJ EC00233
SMOVL C00234 BC00234 V=416.7  +MOVJ EC00234
SMOVL C00235 BC00235 V=416.7  +MOVJ EC00235
MACRO1 MJ#(0) ARGF14
SFTON3D P030
SMOVL C00236 BC00236 V=166.7  +MOVJ EC00236
ARCON
SFTON3D P031
SMOVL C00237 BC00237 V=10.0  +MOVJ EC00237
SMOVL C00238 BC00238 V=10.0  +MOVJ EC00238
ARCOF
SMOVL C00239 BC00239 V=250.0  +MOVJ EC00239
SFTOF3D
SMOVL C00240 BC00240 V=416.7  +MOVJ EC00240
SMOVL C00241 BC00241 V=833.3  +MOVJ EC00241
MOVJ C00242 BC00242 VJ=100.00  +MOVJ EC00242 VJ=100.00
MOVJ C00243 BC00243 VJ=100.00  +MOVJ EC00243 VJ=100.00
'obrot
MOVJ C00244 BC00244 VJ=100.00  +MOVJ EC00244 VJ=100.00
MOVJ C00245 BC00245 VJ=100.00  +MOVJ EC00245 VJ=100.00
'
MOVJ C00246 BC00246 VJ=100.00  +MOVJ EC00246 VJ=100.00
END
